/// machine data that is used through most sequences of the unit (motor speed, axes positions, ...)
TYPE XyTableDataMachine :
STRUCT
  Slowspeed : LREAL;
  Highspeed : LREAL;
END_STRUCT
END_TYPE

(* stored: Version 1.1.0.1
   DUT XyTableDataMachine: Id {39b766e0-2041-42fd-b4f7-17466fd3efc4} *)
